VAR_GLOBAL
	nTime			: ULINT; // Beckhoff specific; Returning The timestamp is a 64-bit integer value, with an accuracy of 100 ns
END_VAR

(* stored: Version 1.1.0.1, ProductVersion 3.1.4024.15
   GVL GVL_System: Id {966d70b5-66fd-4eda-a91e-2962d74a711e} *)
